# EPICS autosave request: utcaApp/Db/fofb_channel.req
file "fofb_processing_channel.req", S=${S}, RTM_CHAN=${RTM_CHAN}
file "fofb_shaper_filt_channel.req", S=${S}, RTM_CHAN=${RTM_CHAN}
file "rtmlamp_channel.req", S=${S}, RTM_CHAN=${RTM_CHAN}
